(* CODESYS project Counter_Lamp.project

Project tree, tasks and I/O mapping:
  Device : CODESYS Control Win V3, 3S - Smart Software Solutions GmbH, version 3.5.12.10
    application Application
      libraries: Standard, * (System)
      task MainTask (cyclic, interval t#20ms, priority 1) calls PLC_PRG
      task VISU_TASK (cyclic, interval 100 ms, priority 31) calls VisuElems.Visu_Prg
      program PLC_PRG [LD]
      visualisation Visualization
  text list GlobalTextList
*)

// Device/Application/PLC_PRG
PROGRAM PLC_PRG
VAR
	
	LIGHT: BOOL;
	START: BOOL;
	SYS: BOOL;
	STOP: BOOL;
	TON1: TON;
	elapsedtime1: TIME;
	LIGHT2: BOOL;
	elapsedtime2: TIME;
	TON2: TON;
	MAINLIGHT: BOOL;
	CTD1: CTD;
	currentValue: WORD;
	maxCount: WORD := 5;
	LoadVar: BOOL;
	Counter: CTU;
	resetButton: BOOL;
END_VAR

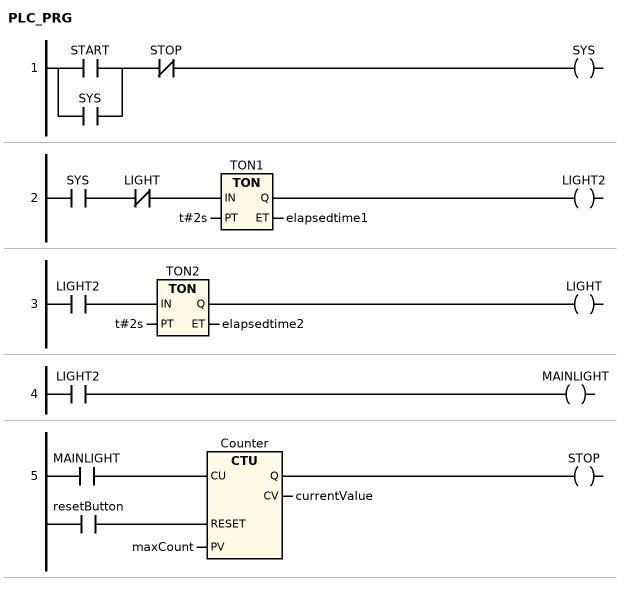
// NETWORK 1
SYS := (START OR SYS) AND NOT STOP;

// NETWORK 2
TON1(IN := SYS AND NOT LIGHT, PT := t#2s, ET => elapsedtime1); // TON
LIGHT2 := TON1.Q;

// NETWORK 3
TON2(IN := LIGHT2, PT := t#2s, ET => elapsedtime2); // TON
LIGHT := TON2.Q;

// NETWORK 4
MAINLIGHT := LIGHT2;

// NETWORK 5
Counter(CU := MAINLIGHT, RESET := resetButton, PV := maxCount, CV => currentValue); // CTU
STOP := Counter.Q;

END_PROGRAM

// Device/Application/Visualization
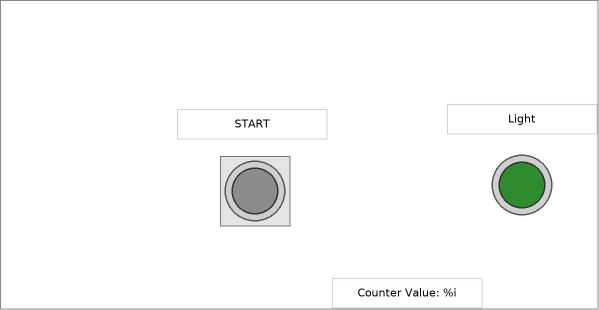
VISUALIZATION Visualization  // 599x310
    PushSwitch (220,156 70x70), variable: PLC_PRG.START, behaviour: TOGGLE, style: Switch-PushSwitch-Gray
    Lamp1 (487,150 70x70), variable: PLC_PRG.MAINLIGHT, style: Lamp-Lamp1-Green
    Textfield (447,104 150x30), "Light"
    Textfield (177,109 150x30), "START"
    Textfield (332,278 150x30), "Counter Value: %i", text variable: PLC_PRG.currentValue
END_VISUALIZATION
